INTERFACE ITF_BaseMainComponent_HMI

END_INTERFACE

(* stored: Version 1.1.0.1
   Itf ITF_BaseMainComponent_HMI: Id {02116d65-3c4f-0345-19e7-8c8d9b7515ea} *)
